// TIA Portal V17 export
// export: Created 2024-08-29T18:23:50.1947352Z, ExportSetting WithDefaults, DisplayName Totally Integrated Automation Portal, DisplayVersion V17 Update 7, DisplayName TIA Portal Openness, DisplayVersion V17 Update 7, DisplayName TIA Portal Version Control Interface, DisplayVersion V17, DisplayName SINAMICS Startdrive Advanced, DisplayVersion V17 SP2, DisplayName SINAMICS Startdrive G110M, G120, G120C, G120D, G120P, G115D, DisplayVersion V17 SP2, DisplayName SINAMICS Startdrive G130, G150, S120, S150, SINAMICS MV, S210, DisplayVersion V17 SP2, DisplayName STEP 7 Professional, DisplayVersion V17 Update 7, DisplayName STEP 7 Safety, DisplayVersion V17 Update 6, DisplayName WinCC Advanced / Unified PC, DisplayVersion V17 Update 7
VAR_GLOBAL   // PLC tag table "pulses"
   hmiPulseInt AT %MD2000 : DInt;
   HMICycleCounterRestartPulse AT %M2004.4 : Bool;
   mode01SelectedPulse AT %M2004.6 : Bool;
   model02SelectedPulse AT %M2004.7 : Bool;
   model03SelectedPulse AT %M2005.0 : Bool;
   model04SelectedPulse AT %M2005.1 : Bool;
   model05SelectedPulse AT %M2005.2 : Bool;
   model06SelectedPulse AT %M2005.3 : Bool;
   model07SelectedPulse AT %M2005.4 : Bool;
   model08SelectedPulse AT %M2005.5 : Bool;
   model09SelectedPulse AT %M2005.6 : Bool;
   model10SelectedPulse AT %M2005.7 : Bool;
   model11SelectedPulse AT %M2006.0 : Bool;
   model12SelectedPulse AT %M2006.1 : Bool;
   model13SelectedPulse AT %M2006.2 : Bool;
   model14SelectedPulse AT %M2006.3 : Bool;
   model15SelectedPulse AT %M2006.4 : Bool;
   alarmPresentPulse AT %M2004.3 : Bool;
   "1stShiftChangePulse" AT %M2004.0 : Bool;
   "2ndShiftChangePulse" AT %M2004.1 : Bool;
   "3rdShiftChangePulse" AT %M2004.2 : Bool;
   stepChangeTimerResetInputPulse AT %M2009.4 : Bool;
   stepChangeTimerResetOutputPulse AT %M2009.5 : Bool;
   stationTurnedOffInSequencePulse AT %M2009.3 : Bool;
   model32SelectedPulse AT %M2008.5 : Bool;
   model31SelectedPulse AT %M2008.4 : Bool;
   model30SelectedPulse AT %M2008.3 : Bool;
   model29SelectedPulse AT %M2008.2 : Bool;
   model27SelectedPulse AT %M2008.0 : Bool;
   model28SelectedPulse AT %M2008.1 : Bool;
   model26SelectedPulse AT %M2007.7 : Bool;
   model25SelectedPulse AT %M2007.6 : Bool;
   model24SelectedPulse AT %M2007.5 : Bool;
   model23SelectedPulse AT %M2007.4 : Bool;
   model22SelectedPulse AT %M2007.3 : Bool;
   model21SelectedPulse AT %M2007.2 : Bool;
   model20SelectedPulse AT %M2007.1 : Bool;
   model19SelectedPulse AT %M2007.0 : Bool;
   model18SelectedPulse AT %M2006.7 : Bool;
   model17SelectedPulse AT %M2006.6 : Bool;
   model16SelectedPulse AT %M2006.5 : Bool;
   scanner3DataLogPulse AT %M2009.2 : Bool;
   scanner2DataLogPulse AT %M2009.1 : Bool;
   scanner1DataLogPulse AT %M2009.0 : Bool;
   motorScannerPulse AT %M2008.6 : Bool;
   rightTrackScannerPulse AT %M2008.7 : Bool;
   leftTrackScannerPulse AT %M2004.5 : Bool;
   scannerOk1Pulse AT %M2009.6 : Bool;
   scannerOk2Pulse AT %M2009.7 : Bool;
   scannerOk3Pulse AT %M2010.0 : Bool;
   leftTrackNokAlarmPulse AT %M2010.1 : Bool;
   rightTrackNokAlarmPulse AT %M2010.2 : Bool;
END_VAR
